// TIA Portal V19 export
ORGANIZATION_BLOCK "Main_1"   // OB201, LAD, ProgramCycle
TITLE = "Main Program Sweep (Cycle)"
// stored: AutoNumber false, IsIECCheckEnabled true, SetENOAutomatically true
   VAR_INPUT
      Initial_Call : Bool;   // Initial call of this OB
      Remanence : Bool;   // =True, if remanent data are available
   END_VAR
   VAR_TEMP   // added for the SCL form of the ladder/FBD networks
      _w1 : Bool;
      _w2 : Bool;
   END_VAR
BEGIN

REGION Network 1: First Cycle
   // Set bit to true in first cycle, and false in all other cycles
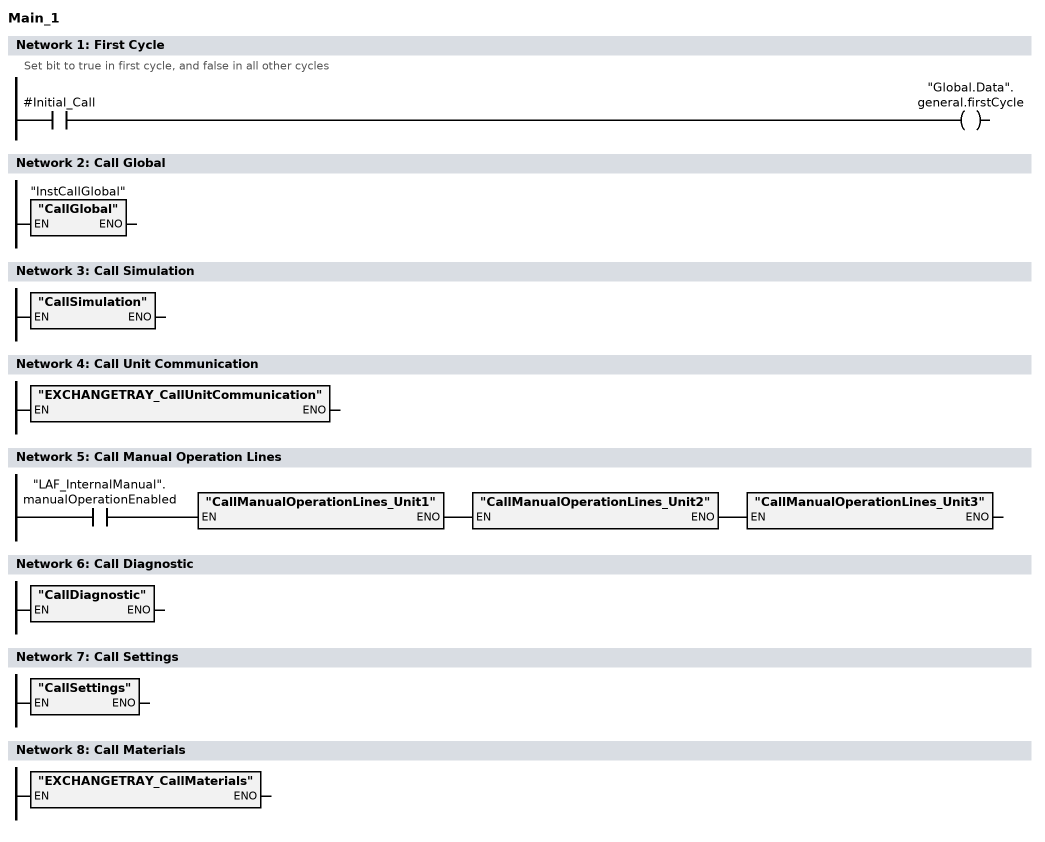
   RUNG wire#powerrail
      Contact( #Initial_Call )
      Coil( "Global.Data".general.firstCycle )
   END_RUNG
   // the same network as SCL:
   "Global.Data".general.firstCycle := #Initial_Call;
END_REGION

REGION Network 2: Call Global
   RUNG wire#powerrail
      "InstCallGlobal"()
   END_RUNG
   // the same network as SCL:
   "InstCallGlobal"();   // "CallGlobal"
END_REGION

REGION Network 3: Call Simulation
   RUNG wire#powerrail
      "CallSimulation"()
   END_RUNG
   // the same network as SCL:
   "CallSimulation"();
END_REGION

REGION Network 4: Call Unit Communication
   RUNG wire#powerrail
      "EXCHANGETRAY_CallUnitCommunication"()
   END_RUNG
   // the same network as SCL:
   "EXCHANGETRAY_CallUnitCommunication"();
END_REGION

REGION Network 5: Call Manual Operation Lines
   RUNG wire#powerrail
      Contact( "LAF_InternalManual".manualOperationEnabled )
      "CallManualOperationLines_Unit1"()
      "CallManualOperationLines_Unit2"()
      "CallManualOperationLines_Unit3"()
   END_RUNG
   // the same network as SCL:
   "CallManualOperationLines_Unit1"(EN := "LAF_InternalManual".manualOperationEnabled, ENO => #_w1);
   "CallManualOperationLines_Unit2"(EN := #_w1, ENO => #_w2);
   IF #_w2 THEN "CallManualOperationLines_Unit3"(); END_IF;
END_REGION

REGION Network 6: Call Diagnostic
   RUNG wire#powerrail
      "CallDiagnostic"()
   END_RUNG
   // the same network as SCL:
   "CallDiagnostic"();
END_REGION

REGION Network 7: Call Settings
   RUNG wire#powerrail
      "CallSettings"()
   END_RUNG
   // the same network as SCL:
   "CallSettings"();
END_REGION

REGION Network 8: Call Materials
   RUNG wire#powerrail
      "EXCHANGETRAY_CallMaterials"()
   END_RUNG
   // the same network as SCL:
   "EXCHANGETRAY_CallMaterials"();
END_REGION
END_ORGANIZATION_BLOCK
